// TwinCAT 3 PLC project ModbusPLC
// ProgramVersion: 3.1.4024.0
// libraries:
//   Tc2_ModbusRTU, * (Beckhoff Automation GmbH)
//   Tc2_Standard, * (Beckhoff Automation GmbH)
//   Tc2_System, * (Beckhoff Automation GmbH)
//   Tc3_Module, * (Beckhoff Automation GmbH)
// project tree:
//   / PlcTask.TcTTO
//   POUs/ MAIN.TcPOU, P_ModbusMaster.TcPOU, P_ModbusSlave.TcPOU
// real-time tasks:
//   TASK PlcTask: cycle T#4ms, priority 20, ADS port 350
// I/O:
//   DEVICE Device 1 (EtherCAT), AmsNetId 5.59.222.134.2.1
//     Term 1 (EK1200) [EK1200-5000 EtherCAT Power supply (2A E-Bus)]
//       Term 2 (EL6022) [EL6022 Interface 2Ch. (RS422/485)]
//       Term 3 (EL9011) [EL9011 End Terminal]
// variable links:
//   ModbusPLC/ModbusPLC Instance <-> Device 1 (EtherCAT)/Term 1 (EK1200)/Term 2 (EL6022)
//     PlcTask Inputs/P_ModbusMaster.MB.InData/D <-> COM Inputs Channel 1/Data In 0
//     PlcTask Inputs/P_ModbusMaster.MB.InData/D @bit {8..168 step 8} <-> COM Inputs Channel 1/Data In {1..21}  (21 links)
//     PlcTask Inputs/P_ModbusMaster.MB.InData/Status <-> COM Inputs Channel 1/Status
//     PlcTask Inputs/P_ModbusSlave.MB.InData/D <-> COM Inputs Channel 2/Data In 0
//     PlcTask Inputs/P_ModbusSlave.MB.InData/D @bit {8..168 step 8} <-> COM Inputs Channel 2/Data In {1..21}  (21 links)
//     PlcTask Inputs/P_ModbusSlave.MB.InData/Status <-> COM Inputs Channel 2/Status
//     PlcTask Outputs/P_ModbusMaster.MB.OutData/Ctrl <-> COM Outputs Channel 1/Ctrl
//     PlcTask Outputs/P_ModbusMaster.MB.OutData/D <-> COM Outputs Channel 1/Data Out 0
//     PlcTask Outputs/P_ModbusMaster.MB.OutData/D @bit {8..168 step 8} <-> COM Outputs Channel 1/Data Out {1..21}  (21 links)
//     PlcTask Outputs/P_ModbusSlave.MB.OutData/Ctrl <-> COM Outputs Channel 2/Ctrl
//     PlcTask Outputs/P_ModbusSlave.MB.OutData/D <-> COM Outputs Channel 2/Data Out 0
//     PlcTask Outputs/P_ModbusSlave.MB.OutData/D @bit {8..168 step 8} <-> COM Outputs Channel 2/Data Out {1..21}  (21 links)

CONFIGURATION ModbusPLC
    RESOURCE PLC ON TwinCAT3
        TASK PlcTask(INTERVAL := T#4ms, PRIORITY := 20);
        PROGRAM MAIN WITH PlcTask : MAIN;
    END_RESOURCE
END_CONFIGURATION

// ---- POUs/MAIN.TcPOU
PROGRAM MAIN
VAR
	
END_VAR

P_ModbusMaster();
P_ModbusSlave();

END_PROGRAM

// ---- POUs/P_ModbusMaster.TcPOU
PROGRAM P_ModbusMaster
VAR
	MB 						: ModbusRtuMaster_KL6x22B;	// change to ModbusRtuMaster_PcCom in case of COM Port
	State					: UINT;
	nLastErrorState			: UINT;
	nLastError				: MODBUS_ERRORS;
	arrRegs					: ARRAY[0..9] OF WORD;
	arrRegs2				: ARRAY[0..9] OF WORD;
	arrCoils				: ARRAY[0..9] OF WORD;
	arrCoils2				: ARRAY[0..9] OF WORD;
	arrInputs				: ARRAY[0..9] OF WORD;
END_VAR

CASE State OF
	
	0:	(*initialization*)
		MB(Execute:=FALSE);
		State:=State+10;
		
	10: (*Reading registers from Outputs or Memory area*)
		(*Function 3(Read Holding Registers)*)
		MB.ReadRegs(
			UnitID:=1 , 								(*Slave address*)
			Quantity:=10 ,								(*Number of data words to be read*)
			MBAddr:=16#4000,							(*Modbus (register) address*)
			cbLength:=20,								(*Size of the data variable used for send or read actions in bytes.*)
			pMemoryAddr:=ADR(arrRegs) ,					(*Address of the variable to which the query result is returned*)
			Execute:=TRUE,
			timeout:=T#1S,
			Error=>);
		
		IF NOT MB.BUSY THEN
			IF NOT MB.Error THEN
				State:=State+10;
			ELSE
				nLastErrorState:=State;
				nLastError:=MB.ErrorId;
				State:=999;
			END_IF
			MB.ReadRegs(Execute:=FALSE);
		END_IF
	
	20:
		(*Writing registers to Outputs or Memory area*)
		(*Function 16(Write Holding Registers) *)	
		MB.WriteRegs(
			UnitID:=1 , 								(*Slave address*)
			Quantity:=10 ,								(*Number of data words to be written*)
			MBAddr:=16#4000,							(*Modbus (register) address*)
			cbLength:=20,								(*Size of the data variable used for send or read actions in bytes.*)
			pMemoryAddr:=ADR(arrRegs2) ,				(*Address of the variable storing the data to be written*)
			Execute:=TRUE,
			timeout:=T#1S,
			Error=>);
		
		IF NOT MB.BUSY THEN
			IF NOT MB.Error THEN
				State:=State+10;
			ELSE
				nLastErrorState:=State;
				nLastError:=MB.ErrorId;
				State:=999;
			END_IF
			MB.WriteRegs(Execute:= FALSE);
		END_IF
	
	30:
		(*Reading bits from Output memory*)
		(*Function 1(Read coils)*)
		MB.ReadCoils(
			UnitID:=1 , 								(*Slave address*)
			Quantity:=SIZEOF(arrCoils)*8 ,				(*Number of data bits to be read*)
			MBAddr:=16#800,								(*Modbus address - Output 16#800*)
			cbLength:=SIZEOF(arrCoils),					(*Size of the data variable used for send or read actions in bytes*)
			pMemoryAddr:=ADR(arrCoils) ,				(*Address of the variable to which the query result is returned*)
			Execute:=TRUE,
			timeout:=T#1S,
			Error=>);
		
		IF NOT MB.BUSY THEN
			IF NOT MB.Error THEN
				State:=State+10;
			ELSE
				nLastErrorState:=State;
				nLastError:=MB.ErrorId;
				State:=999;
			END_IF
			MB.ReadCoils(Execute:=FALSE);
		END_IF
		
	40:
		(*Writing bits to Outputs area*)
		(*Function 15(Write Multiple Coils)*)
		MB.WriteMultipleCoils(
			UnitID:=1 , 								(*Slave address*)
			Quantity:=SIZEOF(arrCoils2)*8 ,				(*Number of data bits to be written*)
			MBAddr:=16#800,								(*Modbus address - Output 16#800*)
			cbLength:=SIZEOF(arrCoils2),				(*Size of the data variable used for send or read actions in bytes*)
			pMemoryAddr:=ADR(arrCoils2) ,				(*Address of the variable storing the data to be written*)
			Execute:=TRUE,
			timeout:=T#1S,
			Error=>);
		
		IF NOT MB.BUSY THEN
			IF NOT MB.Error THEN
				State:=State+10;
			ELSE
				nLastErrorState:=State;
				nLastError:=MB.ErrorId;
				State:=999;
			END_IF
			MB.WriteMultipleCoils(Execute:=FALSE);
		END_IF
		
	50:
		(*Reading registers from Inputs area*)
		(*Function 4(Read Input Registers)*)
		MB.ReadInputRegs(
			UnitID:=1 , 								(*Slave address*)
			Quantity:=10 ,								(*Number of data words to be read*)
			MBAddr:=16#0	,							(*Modbus (register) address*)
			cbLength:=20,								(*Size of the data variable used for send or read actions in bytes.*)
			pMemoryAddr:=ADR(arrInputs) ,				(*Address of the variable to which the query result is returned*)
			Execute:=TRUE,
			timeout :=T#1S,
			Error=> );
		
		IF NOT MB.BUSY THEN
			IF NOT MB.Error THEN
				State:=0;
			ELSE
				nLastErrorState:=State;
				nLastError:=MB.ErrorId;
				State:=999;
			END_IF
			MB.ReadInputRegs(Execute:=FALSE);
		END_IF
			
		999:(*Error handling - subject for modification*) 
			MB(Execute:=FALSE);
			State:=0;
			
			
END_CASE

END_PROGRAM

// ---- POUs/P_ModbusSlave.TcPOU
PROGRAM P_ModbusSlave
VAR
	arrInput	: ARRAY[0..19] OF WORD;
	arrOutput	: ARRAY[0..19] OF WORD;
	arrMemory	: ARRAY[0..19] OF WORD;
	MB			: ModbusRtuSlave_KL6x22B;
END_VAR

MB(
	UnitID:=1 ,
	AdrInputs:= ADR(arrInput),
	SizeInputBytes:=SIZEOF(arrInput) ,
	AdrOutputs:=ADR(arrOutput) ,
	SizeOutputBytes:=SIZEOF(arrOutput) ,
	AdrMemory:=ADR(arrMemory) ,
	SizeMemoryBytes:=SIZEOF(arrMemory) ,
	ErrorId=> );

END_PROGRAM
